(* IEC 61131-3 sources: volt/packages/volt-lsp-iec/test-corpus/bakon-nano/Device/Plc Logic/Application/Library Manager/CmpIecTask, 40 files *)

(* ---- EVTPARAM_CMPIECTASK.dut ---- *)
TYPE EVTPARAM_CMPIECTASK :
STRUCT
	PTASKDESC : POINTER TO Task_Desc;
END_STRUCT
END_TYPE

(* ---- EVTPARAM_CMPIECTASK2.dut ---- *)
TYPE EVTPARAM_CMPIECTASK2 :
STRUCT
	PTASKDESC : POINTER TO Task_Desc2;
END_STRUCT
END_TYPE

(* ---- EVTPARAM_CMPIECTASK_OMITTEDCYCLECOUNTERS.dut ---- *)
TYPE EVTPARAM_CMPIECTASK_OMITTEDCYCLECOUNTERS :
STRUCT
	PTASKDESC : POINTER TO Task_Desc;
	OMITTEDCYCLECOUNTERS : IecTaskOmittedCycleCounters;
END_STRUCT
END_TYPE

(* ---- IEC_CYCLE_STRUCT.dut ---- *)
TYPE IEC_CYCLE_STRUCT :
STRUCT
	PTASKINFO : POINTER TO Task_Info2;
	PAPPLICATION : POINTER TO APPLICATION;
	HTASKHANDLE : RTS_IEC_HANDLE;
END_STRUCT
END_TYPE

(* ---- IECTASKOMITTEDCYCLECOUNTERS.dut ---- *)
TYPE IECTASKOMITTEDCYCLECOUNTERS :
STRUCT
	OMITTEDCYCLES : DWORD;
	CONSECUTIVEOMITTEDCYCLES : DWORD;
END_STRUCT
END_TYPE

(* ---- JITTER_DISTRIBUTION.dut ---- *)
TYPE JITTER_DISTRIBUTION :
STRUCT
	WRANGEMAX : WORD;
	WCOUNTJITTERNEG : WORD;
	WCOUNTJITTERPOS : WORD;
END_STRUCT
END_TYPE

(* ---- TASK_DESC.dut ---- *)
TYPE TASK_DESC :
STRUCT
	UDIID : UDINT;
	UDIDEBUGGINGACTIVEINCYCLE : UDINT;
	HSLOTPOUPOOL : RTS_IEC_HANDLE;
	HIECTASK : RTS_IEC_HANDLE;
	HSCHED : RTS_IEC_HANDLE;
	PAPP : POINTER TO APPLICATION;
	PINFO : POINTER TO Task_Info;
END_STRUCT
END_TYPE

(* ---- TASK_DESC2.dut ---- *)
TYPE TASK_DESC2 :
STRUCT
	UDIID : UDINT;
	UDIDEBUGGINGACTIVEINCYCLE : UDINT;
	HSLOTPOUPOOL : RTS_IEC_HANDLE;
	HIECTASK : RTS_IEC_HANDLE;
	HSCHED : RTS_IEC_HANDLE;
	PAPP : POINTER TO APPLICATION;
	PINFO : POINTER TO Task_Info2;
END_STRUCT
END_TYPE

(* ---- TASK_INFO.dut ---- *)
TYPE TASK_INFO :
STRUCT
	DWVERSION : DWORD;
	PSZNAME : POINTER TO STRING;
	NPRIORITY : INT;
	KINDOFTASK : INT;
	BWATCHDOG : BOOL;
	BPROFILING : BOOL;
	DWEVENTFUNCTIONPOINTER : DWORD;
	PSZEXTERNALEVENT : POINTER TO STRING;
	DWTASKENTRYFUNCTIONPOINTER : DWORD;
	DWWATCHDOGSENSITIVITY : DWORD;
	TINTERVAL : TIME;
	TWATCHDOGTIME : TIME;
	TCYCLETIME : TIME;
	TAVERAGECYCLETIME : TIME;
	TMAXCYCLETIME : TIME;
	TMINCYCLETIME : TIME;
	IJITTER : DINT;
	IJITTERMIN : DINT;
	IJITTERMAX : DINT;
	DWCYCLECOUNT : DWORD;
	ISTATE : WORD;
	WNUMOFJITTERDISTRIBUTIONS : WORD;
	PJITTERDISTRIBUTION : POINTER TO Jitter_Distribution;
END_STRUCT
END_TYPE

(* ---- TASK_INFO2.dut ---- *)
TYPE TASK_INFO2 :
STRUCT
	DWVERSION : DWORD;
	PSZNAME : POINTER TO STRING;
	NPRIORITY : INT;
	KINDOFTASK : INT;
	BWATCHDOG : BOOL;
	BPROFILING : BOOL;
	DWEVENTFUNCTIONPOINTER : POINTER TO BYTE;
	PSZEXTERNALEVENT : POINTER TO STRING;
	DWTASKENTRYFUNCTIONPOINTER : POINTER TO BYTE;
	DWWATCHDOGSENSITIVITY : DWORD;
	DWINTERVAL : DWORD;
	DWWATCHDOGTIME : DWORD;
	DWCYCLETIME : DWORD;
	DWAVERAGECYCLETIME : DWORD;
	DWMAXCYCLETIME : DWORD;
	DWMINCYCLETIME : DWORD;
	IJITTER : DINT;
	IJITTERMIN : DINT;
	IJITTERMAX : DINT;
	DWCYCLECOUNT : DWORD;
	ISTATE : WORD;
	WNUMOFJITTERDISTRIBUTIONS : WORD;
	PJITTERDISTRIBUTION : POINTER TO Jitter_Distribution;
	BTIMESLICING : BOOL;
	BYDUMMY : BYTE;
	WDUMMY : WORD;
	DWIECCYCLECOUNT : DWORD;
END_STRUCT
END_TYPE

(* ---- TASK_WATCHDOGHITCOUNT.dut ---- *)
TYPE TASK_WATCHDOGHITCOUNT :
STRUCT
	DWCONSECUTIVEMAX : DWORD;
	DWTOTAL : DWORD;
END_STRUCT
END_TYPE

(* ---- EVENTIDS.gvl ---- *)
VAR_GLOBAL
	CMPNAME_CMPIECTASK : STRING := 'CmpIecTask';
	CMPID_CMPIECTASK : DWORD := 16#11;
	EVTPARAMID_CMPIECTASK : WORD := 16#1;
	EVTVERSION_CMPIECTASK : WORD := 16#1;
	EVTPARAMID_CMPIECTASK_OMITTEDCYCLECOUNTERS : WORD := 16#2;
	EVTVERSION_CMPIECTASK_OMITTEDCYCLECOUNTERS : WORD := 16#1;
	EVT_AFTERREADINGINPUTS : DWORD := 16#10001;
	EVT_BEFOREWRITINGOUTPUTS : DWORD := 16#10002;
	EVT_BEFOREREADINGINPUTS : DWORD := 16#10003;
	EVT_AFTERWRITINGOUTPUTS : DWORD := 16#10004;
	EVT_IECTASK_RELOADINIT : DWORD := 16#10005;
	EVT_IECTASKCREATEDONE : DWORD := 16#10006;
	EVT_IECTASKPREPAREDELETE : DWORD := 16#10007;
	EVT_IECTASKDEBUGLOOP : DWORD := 16#10008;
	EVT_IECTASKOMITTEDCYCLECOUNTERS : DWORD := 16#10009;
END_VAR

(* ---- SETTINGS.gvl ---- *)
VAR_GLOBAL
	IECTASK_SETTG_KEY_SYNCTASK_NAME_PREFIX : STRING := 'SyncTask';
	IECTASK_SETTG_KEY_SYNCTASK_NAME : STRING := 'Name';
	IECTASK_SETTG_KEY_SYNCTASK_TIMESTAMP : STRING := 'Timestamp';
	IECTASK_SETTG_KEY_SYNCTASK_TYPE : STRING := 'Type';
	IECTASK_SETTG_VALUE_TYPE_APPLICATION : STRING := 'Application';
END_VAR

(* ---- TASKSTATE.gvl ---- *)
VAR_GLOBAL
	TS_NOT_CREATED : WORD := 16#0;
	TS_VALID : WORD := 16#1;
	TS_ACTIVE : WORD := 16#2;
	TS_SUSPENDED : WORD := 16#4;
	TS_DELETED : WORD := 16#8;
	TS_EXCEPTION : WORD := 16#10;
	TS_WATCHDOG_ENABLE : WORD := 16#40;
	TS_DISABLE_TASK_TIME : WORD := 16#80;
	TS_ACTIVATED : WORD := 16#100;
	TS_TOACTIVATE : WORD := 16#200;
	TS_STOP : WORD := 16#400;
	TS_HALT_ON_BP : WORD := 16#800;
	TS_SINGLE_CYCLE : WORD := 16#1000;
	TS_WATCHDOG_ENABLE2 : WORD := 16#2000;
END_VAR

(* ---- TASKTYPE.gvl ---- *)
VAR_GLOBAL
	TASKCYCLIC : INT := 16#0;
	TASKEVENT : INT := 16#1;
	TASKEXTERNAL : INT := 16#2;
	TASKFREEWHEELING : INT := 16#3;
END_VAR

(* ---- TIMEOUT.gvl ---- *)
VAR_GLOBAL
	RTS_TIMEOUT_INFINITE : DINT := -1;
	RTS_TIMEOUT_DEFAULT : DINT := -2;
	RTS_TIMEOUT_NO_WAIT : DINT := 0;
END_VAR

(* ---- VERSION.gvl ---- *)
VAR_GLOBAL
	CMPIECTASK_VERSION_3_4_4_0 : DWORD := 16#3040400;
END_VAR

(* ---- IECTASKCREATE.pou ---- *)
FUNCTION IECTASKCREATE : RTS_IEC_HANDLE
VAR_INPUT
	PAPP : POINTER TO APPLICATION;
	PTASKINFO : POINTER TO Task_Info2;
	PRESULT : POINTER TO RTS_IEC_RESULT;
END_VAR
END_FUNCTION

(* ---- IECTASKCREATE2.pou ---- *)
FUNCTION IECTASKCREATE2 : RTS_IEC_HANDLE
VAR_INPUT
	PAPP : POINTER TO APPLICATION;
	PTASKINFO : POINTER TO Task_Info2;
	PSTASKGROUP : REFERENCE TO STRING;
	PRESULT : POINTER TO RTS_IEC_RESULT;
END_VAR
END_FUNCTION

(* ---- IECTASKDELETE2.pou ---- *)
FUNCTION IECTASKDELETE2 : RTS_IEC_RESULT
VAR_INPUT
	HIECTASK : RTS_IEC_HANDLE;
	ULTIMEOUTMS : UDINT;
END_VAR
END_FUNCTION

(* ---- IECTASKDELETE3.pou ---- *)
FUNCTION IECTASKDELETE3 : RTS_IEC_RESULT
VAR_INPUT
	HIECTASK : RTS_IEC_HANDLE;
	ULTIMEOUTMS : UDINT;
END_VAR
VAR_IN_OUT
	ASYNCSTATE : UDINT;
	FINALRESULT : RTS_IEC_RESULT;
END_VAR
END_FUNCTION

(* ---- IECTASKDISABLESCHEDULING.pou ---- *)
FUNCTION IECTASKDISABLESCHEDULING : RTS_IEC_RESULT
VAR_INPUT
	HIECTASK : RTS_IEC_HANDLE;
END_VAR
END_FUNCTION

(* ---- IECTASKDISABLEWATCHDOG.pou ---- *)
FUNCTION IECTASKDISABLEWATCHDOG : RTS_IEC_RESULT
VAR_INPUT
	HIECTASK : RTS_IEC_HANDLE;
END_VAR
END_FUNCTION

(* ---- IECTASKDISABLEWATCHDOG2.pou ---- *)
FUNCTION IECTASKDISABLEWATCHDOG2 : RTS_IEC_RESULT
VAR_INPUT
	HIECTASK : RTS_IEC_HANDLE;
END_VAR
END_FUNCTION

(* ---- IECTASKENABLESCHEDULING.pou ---- *)
FUNCTION IECTASKENABLESCHEDULING : RTS_IEC_RESULT
VAR_INPUT
	HIECTASK : RTS_IEC_HANDLE;
END_VAR
END_FUNCTION

(* ---- IECTASKENABLEWATCHDOG.pou ---- *)
FUNCTION IECTASKENABLEWATCHDOG : RTS_IEC_RESULT
VAR_INPUT
	HIECTASK : RTS_IEC_HANDLE;
END_VAR
END_FUNCTION

(* ---- IECTASKENABLEWATCHDOG2.pou ---- *)
FUNCTION IECTASKENABLEWATCHDOG2 : RTS_IEC_RESULT
VAR_INPUT
	HIECTASK : RTS_IEC_HANDLE;
END_VAR
END_FUNCTION

(* ---- IECTASKGETCURRENT.pou ---- *)
FUNCTION IECTASKGETCURRENT : RTS_IEC_HANDLE
VAR_INPUT
	PRESULT : POINTER TO RTS_IEC_RESULT;
END_VAR
END_FUNCTION

(* ---- IECTASKGETDESC.pou ---- *)
FUNCTION IECTASKGETDESC : POINTER TO Task_Desc2
VAR_INPUT
	HIECTASK : RTS_IEC_HANDLE;
END_VAR
END_FUNCTION

(* ---- IECTASKGETFIRST.pou ---- *)
FUNCTION IECTASKGETFIRST : RTS_IEC_HANDLE
VAR_INPUT
	PSZAPPNAME : POINTER TO STRING;
	PRESULT : POINTER TO RTS_IEC_RESULT;
END_VAR
END_FUNCTION

(* ---- IECTASKGETINFO2.pou ---- *)
FUNCTION IECTASKGETINFO2 : POINTER TO Task_Info
VAR_INPUT
	HIECTASK : RTS_IEC_HANDLE;
	PRESULT : POINTER TO RTS_IEC_RESULT;
END_VAR
END_FUNCTION

(* ---- IECTASKGETINFO2_INTERNAL.pou ---- *)
FUNCTION IECTASKGETINFO2_INTERNAL : POINTER TO Task_Info
VAR_INPUT
	HIECTASK : RTS_IEC_HANDLE;
	PRESULT : POINTER TO RTS_IEC_RESULT;
END_VAR
END_FUNCTION

(* ---- IECTASKGETINFO3.pou ---- *)
FUNCTION IECTASKGETINFO3 : POINTER TO Task_Info2
VAR_INPUT
	HIECTASK : RTS_IEC_HANDLE;
	PRESULT : POINTER TO RTS_IEC_RESULT;
END_VAR
END_FUNCTION

(* ---- IECTASKGETNEXT.pou ---- *)
FUNCTION IECTASKGETNEXT : RTS_IEC_HANDLE
VAR_INPUT
	PSZAPPNAME : POINTER TO STRING;
	HPREVIECTASK : RTS_IEC_HANDLE;
	PRESULT : POINTER TO RTS_IEC_RESULT;
END_VAR
END_FUNCTION

(* ---- IECTASKGETOMITTEDCYCLECOUNTERS.pou ---- *)
FUNCTION IECTASKGETOMITTEDCYCLECOUNTERS : RTS_IEC_RESULT
VAR_INPUT
	HIECTASK : RTS_IEC_HANDLE;
END_VAR
VAR_IN_OUT
	OMITTEDCYCLECOUNTERS : IecTaskOmittedCycleCounters;
END_VAR
END_FUNCTION

(* ---- IECTASKGETPROFILING.pou ---- *)
FUNCTION IECTASKGETPROFILING : BOOL
END_FUNCTION

(* ---- IECTASKGETWATCHDOGHITCOUNT.pou ---- *)
FUNCTION IECTASKGETWATCHDOGHITCOUNT : RTS_IEC_RESULT
VAR_INPUT
	HIECTASK : RTS_IEC_HANDLE;
	PWATCHDOGHITCOUNT : POINTER TO Task_WatchdogHitCount;
	WWATCHDOGHITCOUNTSIZE : WORD;
END_VAR
END_FUNCTION

(* ---- IECTASKRELOAD.pou ---- *)
FUNCTION IECTASKRELOAD : RTS_IEC_HANDLE
VAR_INPUT
	HIECTASK : RTS_IEC_HANDLE;
	UDITIMEOUTMS : UDINT;
	PRESULT : POINTER TO RTS_IEC_RESULT;
END_VAR
END_FUNCTION

(* ---- IECTASKRESETSTATISTICS.pou ---- *)
FUNCTION IECTASKRESETSTATISTICS : RTS_IEC_RESULT
VAR_INPUT
	HIECTASK : RTS_IEC_HANDLE;
END_VAR
END_FUNCTION

(* ---- IECTASKSETSTARTOFFSET.pou ---- *)
FUNCTION IECTASKSETSTARTOFFSET : RTS_IEC_RESULT
VAR_INPUT
	SIECTASKNAME : STRING;
	STARTOFFSETUS : DINT;
END_VAR
END_FUNCTION
